// TIA Portal V20 export
DATA_BLOCK "GDB_MovePath"   // DB21
{ S7_Optimized_Access := 'TRUE' }
// stored: MemoryReserve 100
BEGIN
END_DATA_BLOCK
